// Mitsubishi GX Works2 project: 실린더 제어하기2-1 0920   PLC: Q03UDV

PROGRAM MAIN
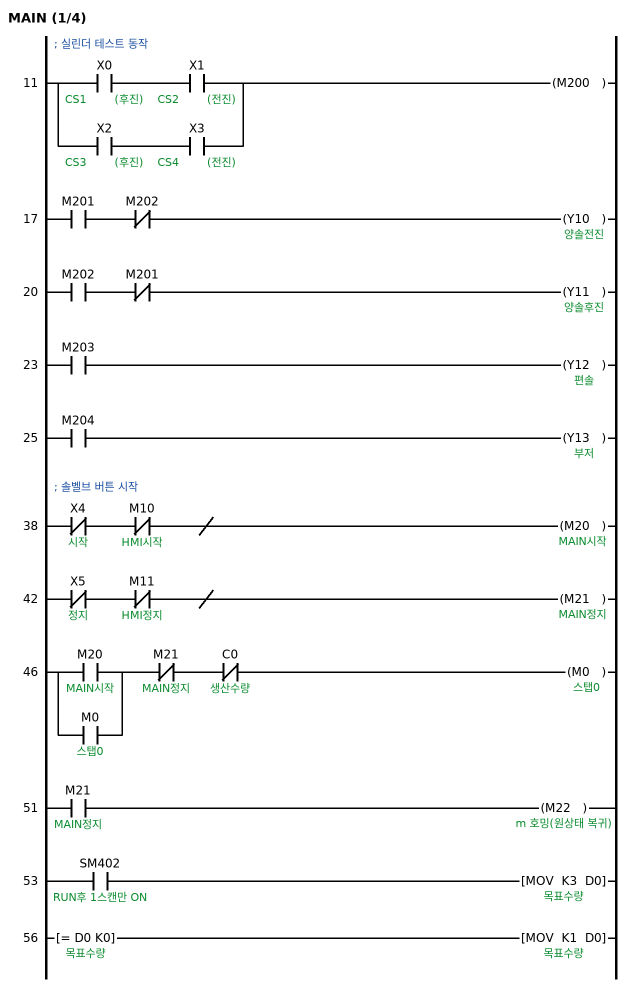
; 실린더 테스트 동작
11    LD      X0  ; CS1        (후진)
      AND     X1  ; CS2        (전진)
      LD      X2  ; CS3        (후진)
      AND     X3  ; CS4        (전진)
      ORB
      OUT     M200
17    LD      M201
      ANI     M202
      OUT     Y10  ; 양솔전진
20    LD      M202
      ANI     M201
      OUT     Y11  ; 양솔후진
23    LD      M203
      OUT     Y12  ; 편솔
25    LD      M204
      OUT     Y13  ; 부저
; 솔벨브 버튼 시작
38    LDI     X4  ; 시작
      ANI     M10  ; HMI시작
      INV
      OUT     M20  ; MAIN시작
42    LDI     X5  ; 정지
      ANI     M11  ; HMI정지
      INV
      OUT     M21  ; MAIN정지
46    LD      M20  ; MAIN시작
      OR      M0  ; 스탭0
      ANI     M21  ; MAIN정지
      ANI     C0  ; 생산수량
      OUT     M0  ; 스탭0
51    LD      M21  ; MAIN정지
      OUT     M22  ; m 호밍(원상태 복귀)
53    LD      SM402  ; RUN후 1스캔만 ON
      MOV     K3 D0  ; 목표수량
56    LD=     D0 K0  ; 목표수량
      MOV     K1 D0
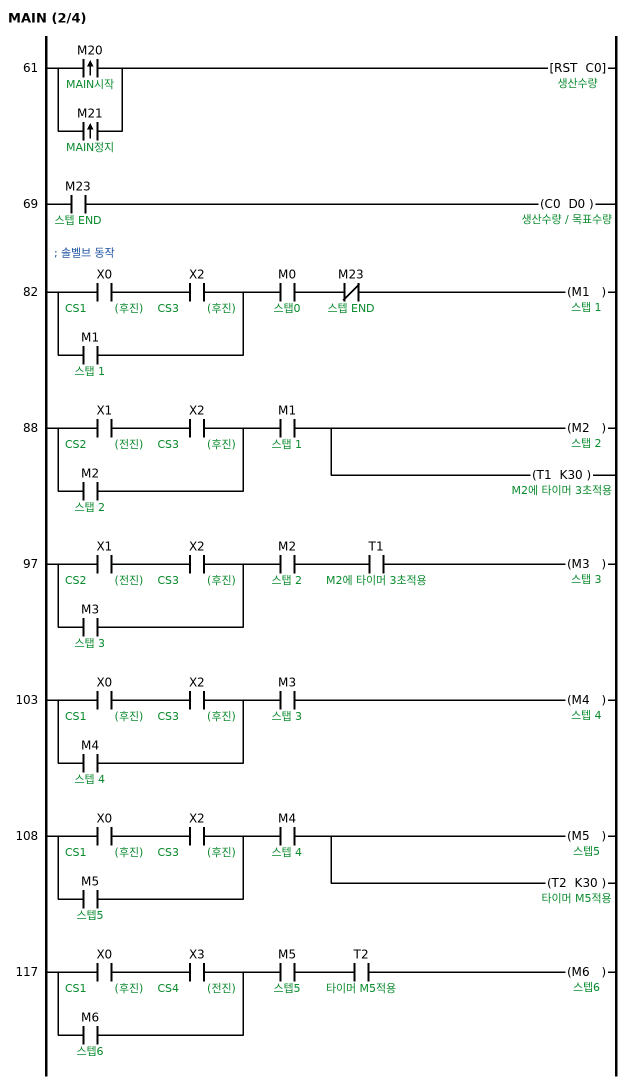
61    LDP     M20  ; MAIN시작
      ORP     M21  ; MAIN정지
      RST     C0  ; 생산수량
69    LD      M23  ; 스텝 END
      OUT     C0 D0  ; 생산수량 / 목표수량
; 솔벨브 동작
82    LD      X0  ; CS1        (후진)
      AND     X2  ; CS3        (후진)
      OR      M1  ; 스탭 1
      AND     M0  ; 스탭0
      ANI     M23  ; 스텝 END
      OUT     M1  ; 스탭 1
88    LD      X1  ; CS2        (전진)
      AND     X2  ; CS3        (후진)
      OR      M2  ; 스탭 2
      AND     M1  ; 스탭 1
      OUT     M2  ; 스탭 2
      OUT     T1 K30  ; M2에 타이머 3초적용
97    LD      X1  ; CS2        (전진)
      AND     X2  ; CS3        (후진)
      OR      M3  ; 스탭 3
      AND     M2  ; 스탭 2
      AND     T1  ; M2에 타이머 3초적용
      OUT     M3  ; 스탭 3
103   LD      X0  ; CS1        (후진)
      AND     X2  ; CS3        (후진)
      OR      M4  ; 스텝 4
      AND     M3  ; 스탭 3
      OUT     M4  ; 스텝 4
108   LD      X0  ; CS1        (후진)
      AND     X2  ; CS3        (후진)
      OR      M5  ; 스텝5
      AND     M4  ; 스텝 4
      OUT     M5  ; 스텝5
      OUT     T2 K30  ; 타이머 M5적용
117   LD      X0  ; CS1        (후진)
      AND     X3  ; CS4        (전진)
      OR      M6  ; 스텝6
      AND     M5  ; 스텝5
      AND     T2  ; 타이머 M5적용
      OUT     M6  ; 스텝6
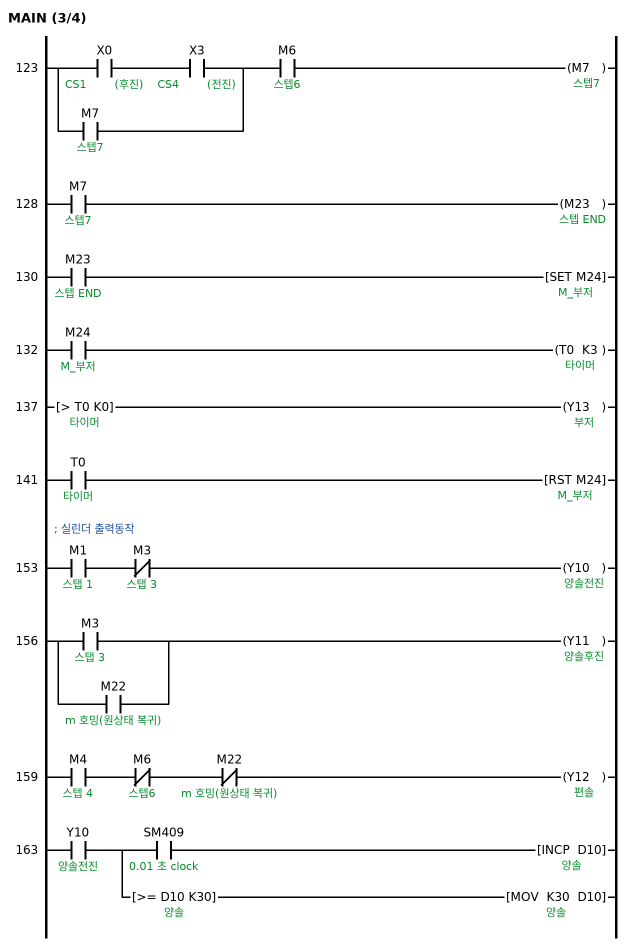
123   LD      X0  ; CS1        (후진)
      AND     X3  ; CS4        (전진)
      OR      M7  ; 스텝7
      AND     M6  ; 스텝6
      OUT     M7  ; 스텝7
128   LD      M7  ; 스텝7
      OUT     M23  ; 스텝 END
130   LD      M23  ; 스텝 END
      SET     M24  ; M_부저
132   LD      M24  ; M_부저
      OUT     T0 K3  ; 타이머
137   LD>     T0 K0  ; 타이머
      OUT     Y13  ; 부저
141   LD      T0  ; 타이머
      RST     M24  ; M_부저
; 실린더 출력동작
153   LD      M1  ; 스탭 1
      ANI     M3  ; 스탭 3
      OUT     Y10  ; 양솔전진
156   LD      M3  ; 스탭 3
      OR      M22  ; m 호밍(원상태 복귀)
      OUT     Y11  ; 양솔후진
159   LD      M4  ; 스텝 4
      ANI     M6  ; 스텝6
      ANI     M22  ; m 호밍(원상태 복귀)
      OUT     Y12  ; 편솔
163   LD      Y10  ; 양솔전진
      MPS
      AND     SM409  ; 0.01 초 clock
      INCP    D10  ; 양솔
      MPP
      AND>=   D10 K30  ; 양솔
      MOV     K30 D10
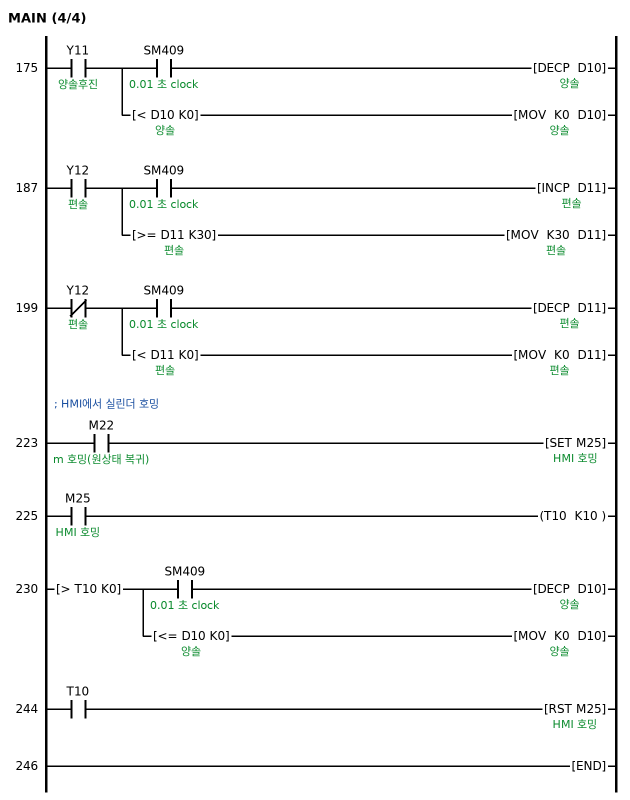
175   LD      Y11  ; 양솔후진
      MPS
      AND     SM409  ; 0.01 초 clock
      DECP    D10
      MPP
      AND<    D10 K0  ; 양솔
      MOV     K0 D10
187   LD      Y12  ; 편솔
      MPS
      AND     SM409  ; 0.01 초 clock
      INCP    D11  ; 편솔
      MPP
      AND>=   D11 K30  ; 편솔
      MOV     K30 D11
199   LDI     Y12  ; 편솔
      MPS
      AND     SM409  ; 0.01 초 clock
      DECP    D11
      MPP
      AND<    D11 K0  ; 편솔
      MOV     K0 D11
; HMI에서 실린더 호밍
223   LD      M22  ; m 호밍(원상태 복귀)
      SET     M25  ; HMI 호밍
225   LD      M25  ; HMI 호밍
      OUT     T10 K10
230   LD>     T10 K0
      MPS
      AND     SM409  ; 0.01 초 clock
      DECP    D10
      MPP
      AND<=   D10 K0  ; 양솔
      MOV     K0 D10
244   LD      T10
      RST     M25  ; HMI 호밍
246   END
END_PROGRAM
